// TwinCAT 3 PLC project PLC
// ProgramVersion: 3.1.4026.15
// CompilerDefines: VISU_USEPROPERTYINFO,VISU_USEWSTRING
// libraries:
//   machine_alarm_manager, * (Beckhoff Automation K.K.)
//   Tc2_MC2, * (Beckhoff Automation GmbH)
//   Tc2_Standard, * (Beckhoff Automation GmbH)
//   Tc2_System, * (Beckhoff Automation GmbH)
//   Tc2_Utilities, * (Beckhoff Automation GmbH)
//   VisuSymbols, 4.5.0.0 (System)
// project tree:
//   DUTs/ AlarmList.TcDUT, AreaStatus.TcDUT
//   / GlobalTextList.TcGTLO, PlcTask.TcTTO, Visualization Manager.TcVMO (not stored), VISU_TASK.TcTTO
//   GVLs/ GVL.TcGVL, Param.TcGVL
//   POUs/ AlarmManager.TcPOU, FB_DelaySampling.TcPOU, FB_MovingAverage.TcPOU, MAIN.TcPOU
//   VISUs/ current.TcVIS, history.TcVIS, languages.TcTLO, main.TcVIS, Visualization.TcVIS
// real-time tasks:
//   TASK PlcTask: cycle T#10ms, priority 20, ADS port 350
//   TASK VISU_TASK: cycle T#100000us, priority 30, ADS port 351
// motion (NC):
//   TASK NC-Task 1 SAF: cycle T#2ms, priority 4, ADS port 501
//   TASK NC-Task 1 SVB: cycle T#10ms, priority 8, ADS port 511
//   AXIS Axis 1 (id 1)
//     General: UnitName=°
//     Dynamic: Acceleration=1769.307, Deceleration=1769.307, Jerk=5307.921
//     Velo: RefSearch=11.79538, RefSync=11.79538, SlowManual=58.9769, FastManual=353.8614, Fast=1179.538, Maximum=1179.538
//     OtherSettings: AllowMotionCmdToSlave=true
//     encoder EncType=19
//       EncPara: ScaleFactorNumerator=360, ScaleFactorDenominator=10485760, MaxCount=#xffffffff
//     drive DrvType=16
//       DrvPara: MaxCount=#xffffffff, DriveControlDWord=#x00020100
//         Analog: VeloReferenz=1297.4918, VeloScale=32, TorqueSetpointScale=10, ScaleFactorActTorque=0.1
//         TimeComp: TaskDelayCycles=1
//     controller CtrType=1
//       CtrPara: PriorControlFactor=1
//         Observer: BandWidth=20
//   AXIS Axis 2 (id 2)
//     General: UnitName=°
//     Dynamic: Acceleration=1769.307, Deceleration=1769.307, Jerk=5307.921
//     Velo: RefSearch=11.79538, RefSync=11.79538, SlowManual=58.9769, FastManual=353.8614, Fast=1179.538, Maximum=1179.538
//     OtherSettings: AllowMotionCmdToSlave=true
//     encoder EncType=19
//       EncPara: ScaleFactorNumerator=360, ScaleFactorDenominator=10485760, MaxCount=#xffffffff
//     drive DrvType=16
//       DrvPara: MaxCount=#xffffffff, DriveControlDWord=#x00020100
//         Analog: VeloReferenz=1297.4918, VeloScale=32, TorqueSetpointScale=10, ScaleFactorActTorque=0.1
//         TimeComp: TaskDelayCycles=1
//     controller CtrType=1
//       CtrPara: PriorControlFactor=1
//         PosDiffControl: Enable=false
//         Observer: BandWidth=20
// I/O:
//   DEVICE Device 2 (EtherCAT), AmsNetId 5.69.67.250.3.1
//     Term 1 (EK1100) [EK1100 EtherCAT Coupler (2A E-Bus)]
//       Term 2 (EL1012) [EL1012 2Ch. Dig. Input 24V, 10µs]
//       Term 3 (EL1004) [EL1004 4Ch. Dig. Input 24V, 3ms]
//       Term 4 (EL1918) [EL1918, 8Ch. Safety Input 24V, TwinSAFE]
//         modules: Module 1 (FSOE), Module 2 (FSLOGIC)
//       Term 5 (EL2004) [EL2004 4Ch. Dig. Output 24V, 0.5A]
//       Term 6 (EL2084) [EL2084 4Ch. Dig. Output 24V, 0.5A, switching to negative]
//       Term 7 (EL5101-0090) [EL5101-0090 1Ch. Inc. Encoder 5V, TwinSAFE SC]
//         modules: Module 1 (EL5101-0090)
//       Term 8 (ELM7212-9018) [ELM7212-9018 2Ch. Servo Terminal (48 V, 4,5 A RMS, OCT, STO, Safe Motion, TwinSAFE Logic)]
//         modules: Module 1 (SAFETY)
//         startup 32785:21 := 0E01 // DRV Motor Settings Ch.1 / Commutation offset
//         startup 32785:27 := 10270000 // DRV Motor Settings Ch.1 / Motor speed limitation
//         startup 28688:11 := F90C // DRV Outputs Ch.1 / Torque limitation
//         startup 32784:19 := FD00 // DRV Amplifier Settings Ch.1 / Current loop proportional gain
//         startup 32784:18 := 0600 // DRV Amplifier Settings Ch.1 / Current loop integral time
//         startup 32784:21 := 2B000000 // DRV Amplifier Settings Ch.1 / Velocity loop proportional gain
//         startup 32784:20 := 96000000 // DRV Amplifier Settings Ch.1 / Velocity loop integral time
//         startup 33041:21 := 0E01 // DRV Motor Settings Ch.2 / Commutation offset
//         startup 33041:27 := 10270000 // DRV Motor Settings Ch.2 / Motor speed limitation
//         startup 28944:11 := F90C // DRV Outputs Ch.2 / Torque limitation
//         startup 33040:19 := FD00 // DRV Amplifier Settings Ch.2 / Current loop proportional gain
//         startup 33040:18 := 0600 // DRV Amplifier Settings Ch.2 / Current loop integral time
//         startup 33040:21 := 2B000000 // DRV Amplifier Settings Ch.2 / Velocity loop proportional gain
//         startup 33040:20 := 96000000 // DRV Amplifier Settings Ch.2 / Velocity loop integral time
//       Term 9 (EL9011) [EL9011 End Terminal]
//   DEVICE Device 1 (EtherCAT Automation Protocol), AmsNetId 5.69.67.250.2.1
//     Box 10 (Publisher)
//     Box 11 (Subscriber)
//     Box 12 (Publisher)
// variable links:
//   Device 2 (EtherCAT) <-> Device 1 (EtherCAT Automation Protocol)/Box 10 (Publisher)
//     Term 1 (EK1100)/Term 8 (ELM7212-9018)/Module 1 (SAFETY)/SAFETY FSoE Connection 3 Send Message/Message_11 <-> Pub-Var-Safety/Outputs/VarData
//   Device 2 (EtherCAT) <-> Device 1 (EtherCAT Automation Protocol)/Box 11 (Subscriber)
//     Term 1 (EK1100)/Term 8 (ELM7212-9018)/Module 1 (SAFETY)/SAFETY FSoE Connection 3 Receive Message/Message_11 <-> Sub-Var-Safety/Inputs/VarData
//   Device 2 (EtherCAT) <-> Device 2 (EtherCAT)/Term 1 (EK1100)/Term 8 (ELM7212-9018)
//     Term 1 (EK1100)/Term 4 (EL1918)/Module 1 (FSOE)/FSoE Inputs/FSOE <-> Module 1 (SAFETY)/SAFETY FSoE Connection 1 Receive Message/Message_3
//     Term 1 (EK1100)/Term 4 (EL1918)/Module 1 (FSOE)/FSoE Outputs/FSOE <-> Module 1 (SAFETY)/SAFETY FSoE Connection 1 Send Message/Message_3
//     Term 1 (EK1100)/Term 7 (EL5101-0090)/Module 1 (EL5101-0090)/TSC Inputs/TSC <-> Module 1 (SAFETY)/SAFETY FSoE Connection 2 Receive Message/Message_4
//     Term 1 (EK1100)/Term 7 (EL5101-0090)/Module 1 (EL5101-0090)/TSC Outputs/TSC <-> Module 1 (SAFETY)/SAFETY FSoE Connection 2 Send Message/Message_4
//   NC-Task 1 SAF/Axes/Axis 1 <-> Device 2 (EtherCAT)/Term 1 (EK1100)/Term 8 (ELM7212-9018)
//     Drive/Inputs/In/nDataIn1 <-> DRV Following error actual value Channel 1/Following error actual value
//     Drive/Inputs/In/nDcOutputTime <-> InfoData/DcOutputShift
//     Drive/Inputs/In/nState1 <-> DRV Statusword Channel 1/Statusword
//     Drive/Inputs/In/nState2 <-> DRV Statusword Channel 1/Statusword @bit 8
//     Drive/Inputs/In/nState4 @bit 1 <-> WcState/InputToggle0
//     Drive/Inputs/In/nState4 <-> WcState/WcState0
//     Drive/Outputs/Out/nCtrl1 <-> DRV Controlword Channel 1/Controlword
//     Drive/Outputs/Out/nCtrl2 <-> DRV Controlword Channel 1/Controlword @bit 8
//     Drive/Outputs/Out/nDataOut1 <-> DRV Target position Channel 1/Target position
//     Enc/Inputs/In/nDataIn1 <-> FB Position Channel 1/Position
//     Enc/Inputs/In/nDcInputTime <-> InfoData/DcInputShift
//     Enc/Inputs/In/nState4 @bit 1 <-> WcState/InputToggle0
//     Enc/Inputs/In/nState4 <-> WcState/WcState0
//   NC-Task 1 SAF/Axes/Axis 2 <-> Device 2 (EtherCAT)/Term 1 (EK1100)/Term 8 (ELM7212-9018)
//     Drive/Inputs/In/nDataIn1 <-> DRV Following error actual value Channel 2/Following error actual value
//     Drive/Inputs/In/nDcOutputTime <-> InfoData/DcOutputShift
//     Drive/Inputs/In/nState1 <-> DRV Statusword Channel 2/Statusword
//     Drive/Inputs/In/nState2 <-> DRV Statusword Channel 2/Statusword @bit 8
//     Drive/Inputs/In/nState4 @bit 1 <-> WcState/InputToggle0
//     Drive/Inputs/In/nState4 <-> WcState/WcState0
//     Drive/Outputs/Out/nCtrl1 <-> DRV Controlword Channel 2/Controlword
//     Drive/Outputs/Out/nCtrl2 <-> DRV Controlword Channel 2/Controlword @bit 8
//     Drive/Outputs/Out/nDataOut1 <-> DRV Target position Channel 2/Target position
//     Enc/Inputs/In/nDataIn1 <-> FB Position Channel 2/Position
//     Enc/Inputs/In/nDcInputTime <-> InfoData/DcInputShift
//     Enc/Inputs/In/nState4 @bit 1 <-> WcState/InputToggle0
//     Enc/Inputs/In/nState4 <-> WcState/WcState0
//   PLC/PLC Instance <-> Device 1 (EtherCAT Automation Protocol)/Box 11 (Subscriber)
//     PlcTask Inputs/MAIN.safety_master_station_emo <-> Sub-Var-Safety/Inputs/VarData/FSoE Data[0]
//   PLC/PLC Instance <-> Device 1 (EtherCAT Automation Protocol)/Box 12 (Publisher)
//     PlcTask Outputs/MAIN.eap_export_information <-> Pub-Var 11/Outputs/VarData
//   PLC/PLC Instance <-> Device 2 (EtherCAT)/Term 1 (EK1100)/Term 2 (EL1012)
//     PlcTask Inputs/MAIN.bWarningSigna02 <-> Channel 1/Input
//     PlcTask Inputs/MAIN.bWarningSigna0l <-> Channel 2/Input
//   PLC/PLC Instance <-> Device 2 (EtherCAT)/Term 1 (EK1100)/Term 3 (EL1004)
//     PlcTask Inputs/MAIN.bMcReset <-> Channel 1/Input
//   PLC/PLC Instance <-> Device 2 (EtherCAT)/Term 1 (EK1100)/Term 4 (EL1918)
//     PlcTask Inputs/MAIN.safety_emo[1] <-> Module 1 (FSOE)/FSoE Inputs/FSOE/FSIN Module 1.Input
//     PlcTask Inputs/MAIN.safety_emo[2] <-> Module 1 (FSOE)/FSoE Inputs/FSOE/FSIN Module 2.Input
//     PlcTask Inputs/MAIN.safety_input_collision_sensor <-> Module 1 (FSOE)/FSoE Inputs/FSOE/FSIN Module 4.Input
//   PLC/PLC Instance <-> Device 2 (EtherCAT)/Term 1 (EK1100)/Term 8 (ELM7212-9018)
//     PlcTask Inputs/MAIN.Enc2ActError <-> Module 1 (SAFETY)/SAFETY Standard Inputdata/Standard Out Var 10
//     PlcTask Inputs/MAIN.Enc2CmdError <-> Module 1 (SAFETY)/SAFETY Standard Inputdata/Standard Out Var 9
//     PlcTask Inputs/MAIN.SafetyMonitorSetSpeed <-> Module 1 (SAFETY)/SAFETY Standard Inputdata/Standard Out Var 14
//     PlcTask Inputs/MAIN.SafetyMonitorSpeed <-> Module 1 (SAFETY)/SAFETY Standard Inputdata/Standard Out Var 12
//     PlcTask Inputs/MAIN.SafetyRefMonitorSpeed <-> Module 1 (SAFETY)/SAFETY Standard Inputdata/Standard Out Var 13
//     PlcTask Outputs/MAIN.bSafetyErrAck <-> Module 1 (SAFETY)/SAFETY Standard Outputdata/Standard In Var 1
//     PlcTask Outputs/MAIN.bSafetyReset <-> Module 1 (SAFETY)/SAFETY Standard Outputdata/Standard In Var 7
//     PlcTask Outputs/MAIN.bSafetyRun <-> Module 1 (SAFETY)/SAFETY Standard Outputdata/Standard In Var 2
//     PlcTask Outputs/MAIN.diSpeedAct <-> Module 1 (SAFETY)/SAFETY Standard Outputdata/Standard In Var 6
//     PlcTask Outputs/MAIN.diSpeedCmd <-> Module 1 (SAFETY)/SAFETY Standard Outputdata/Standard In Var 8
//   PLC/PLC Instance <-> NC-Task 1 SAF/Axes/Axis 1
//     PlcTask Inputs/MAIN.stAxis[1].NcToPlc <-> Outputs/ToPlc
//     PlcTask Outputs/MAIN.stAxis[1].PlcToNc <-> Inputs/FromPlc
//   PLC/PLC Instance <-> NC-Task 1 SAF/Axes/Axis 2
//     PlcTask Inputs/MAIN.stAxis[2].NcToPlc <-> Outputs/ToPlc
//     PlcTask Outputs/MAIN.stAxis[2].PlcToNc <-> Inputs/FromPlc

CONFIGURATION PLC
    RESOURCE PLC ON TwinCAT3
        TASK PlcTask(INTERVAL := T#10ms, PRIORITY := 20);
        TASK VISU_TASK(INTERVAL := T#100000us, PRIORITY := 30);
        PROGRAM MAIN WITH PlcTask : MAIN;
        PROGRAM VisuElems_Visu_Prg WITH VISU_TASK : VisuElems.Visu_Prg;
    END_RESOURCE
END_CONFIGURATION

// ---- DUTs/AlarmList.TcDUT
{attribute 'qualified_only'}
{attribute 'strict'}
{attribute 'to_string'}
TYPE AlarmList :
(
	emergency_stop := 1,
	encoder_error,
	approach,
	proximity,
	collision
);
END_TYPE

// ---- DUTs/AreaStatus.TcDUT
{attribute 'qualified_only'}
{attribute 'strict'}
{attribute 'to_string'}
TYPE AreaStatus :
(
	Safe := 0,
	Hazard := 1,
	Warning_Level1 := 2,
	Warning_Level2 := 3
) := Safe;
END_TYPE

// ---- GVLs/GVL.TcGVL
{attribute 'qualified_only'}
VAR_GLOBAL
	 fb_alarm : ARRAY [1..AlarmEventParam.ALARM_MAX_COUNT] OF POINTER TO FB_Alarm;
END_VAR

// ---- GVLs/Param.TcGVL
{attribute 'qualified_only'}
VAR_GLOBAL CONSTANT
	NumberOfWarningArea		: INT := 2;
END_VAR

// ---- POUs/MAIN.TcPOU
PROGRAM MAIN
VAR
	
	
	stAxis				: ARRAY[1..2] OF AXIS_REF;
	fbMcPower			: ARRAY[1..2] OF MC_Power;
	fbMcReset			: ARRAY[1..2] OF MC_Reset;
	fbMcMoveVelocity	: ARRAY[1..2] OF MC_MoveVelocity;
	fbMcHalt			: ARRAY[1..2] OF MC_Halt;
	
	bPower		: BOOL;
	bRun		: BOOL;
	bStop		: BOOL;
	bMcReset		AT%I*	: BOOL;
	bSafetyReset	AT%Q*	: BOOL;
	bSafetyRun		AT%Q*	: BOOL := TRUE;
	bSafetyErrAck	AT%Q*	: BOOL;
	diSpeedAct		AT%Q*	: DINT;
	diSpeedCmd		AT%Q*	: DINT; 
	
	bWarningSigna0l		AT%I*	: BOOL;
	bWarningSigna02		AT%I*	: BOOL;
	Enc2ActError		AT%I*	: BOOL;
	Enc2CmdError		AT%I*	: BOOL;
	
	lrOverride		: LREAL := 50;
	_override		: LREAL;
	lrVelocity		: LREAL := 360;
	lrGearRate		: LREAL := 10;
	lrIncrement		: LREAL := 1048576;
	lrWheelIncrement	:LREAL;
	lrExtEncoderIncrement		: LREAL := 1000;
	
	diTaskIdx			: DINT;
	udiCycletime		: UDINT;
	udiTimeIntervel		: UDINT;
	udiCycleCount		: UDINT;
	fbDelaySampling		: FB_DelaySampling;
	fbDelaySamplingSet	: FB_DelaySampling;
	
	diPositionAct			: DINT;
	diPositionBufferAct		: DINT;
	diPositionCmd			: DINT;
	diPositionBufferCmd		: DINT;
	
	Mode	: INT;
	i		: UINT;
	//_Mode	: INT;
	//mode_change_delay_timer	: TON := (PT := T#1S);
	
	safety_input_collision_sensor AT%I* : BOOL;
	safety_master_station_emo AT%I* : BOOL;
	safety_emo AT%I* : ARRAY [1..2] OF BOOL;
	
	running_startup_delapy : TON := (PT := T#1S);
	
	eap_export_information	AT%Q* : ARRAY [0..7] OF BOOL;
	
	monitor_speed_average : FB_MovingAverage;
	monitor_refspeed_average : FB_MovingAverage;
	monitor_setspeed_average : FB_MovingAverage;

	SafetyMonitorSpeed AT%I* : DINT;
	SafetyRefMonitorSpeed AT%I* : DINT;
	SafetyMonitorSetSpeed AT%I* : DINT;
	
END_VAR


// Set override speed to 25 while 1sec after motor starting up. Otherwise safety error would occured by speed differential watching.
running_startup_delapy(IN := stAxis[1].Status.Moving);
IF running_startup_delapy.Q THEN
	_override := lrOverride;
ELSE
	_override := 30.0;
END_IF

FOR i:=1 TO 2 DO
	stAxis[i].ReadStatus();
	fbMcPower[i](
	Axis:= stAxis[i], 
	Enable:= bPower, 
	Enable_Positive:= bPower, 
	Enable_Negative:= bPower,
	Override := _override);

	fbMcHalt[i](
		Axis:= stAxis[i], 
		Execute:= bStop, 
		Deceleration:= 3600);
	
	fbMcReset[i](
		Axis:= stAxis[i], 
		Execute:= bMcReset);
	
	fbMcMoveVelocity[i](
		Axis:= stAxis[i],
		Execute:= bRun,
		Velocity:= lrVelocity, 
		//Direction:= MC_Direction.MC_Negative_Direction, 
		BufferMode:= MC_BufferMode.MC_Aborting);	
END_FOR
fbMcMoveVelocity[1].Direction := MC_Direction.MC_Negative_Direction;
fbMcMoveVelocity[2].Direction := MC_Direction.MC_Positive_Direction;

bSafetyReset := bMcReset;
bSafetyErrAck := bMcReset;
IF bMcReset THEN
	Mode := AreaStatus.Safe;
END_IF

IF NOT bWarningSigna0l THEN
	Mode := AreaStatus.Warning_Level1;
	IF NOT bWarningSigna02 THEN
		Mode := AreaStatus.Warning_Level2;
	END_IF
ELSIF (stAxis[1].NcToPlc.ErrorCode <> 0) OR (stAxis[2].NcToPlc.ErrorCode <> 0) THEN
	Mode := AreaStatus.Hazard;
ELSE
	Mode := AreaStatus.Safe;
END_IF

CASE Mode OF

	AreaStatus.Safe:
						lrOverride := 50;	
						
	AreaStatus.Warning_Level1:
						lrOverride := 25;
						
	AreaStatus.Warning_Level2:
						lrOverride := 10;
						
	AreaStatus.Hazard:
						lrOverride := 0;
	
END_CASE


lrWheelIncrement := lrIncrement * lrGearRate / 360;
diPositionAct := LREAL_TO_DINT(-1 * stAxis[1].NcToPlc.ActPos * lrWheelIncrement / lrExtEncoderIncrement);
diSpeedAct := diPositionAct - diPositionBufferAct; 
diPositionCmd := LREAL_TO_DINT(-1 * stAxis[1].NcToPlc.SetPos * lrWheelIncrement / lrExtEncoderIncrement);
diSpeedCmd := diPositionCmd - diPositionBufferCmd; 

diTaskIdx := GETCURTASKINDEXEX();
IF diTaskIdx > 0 THEN
    udiCycleTime := _TaskInfo[diTaskIdx].CycleTime;
	udiCycleCount := (udiTimeIntervel*10000) / udiCycleTime;
END_IF
fbDelaySampling(udiDelaySampling:= udiCycleCount, diData:= diPositionAct, diOutData=> diPositionBufferAct);
fbDelaySamplingSet(udiDelaySampling:= udiCycleCount, diData:= diPositionCmd, diOutData=> diPositionBufferCmd);

// Alarm signal

IF AlarmManager.init THEN
	GVL.fb_alarm[AlarmList.emergency_stop]^.set_activate := NOT safety_master_station_emo OR NOT safety_emo[1] OR NOT safety_emo[2];
	GVL.fb_alarm[AlarmList.approach]^.set_activate := Mode = AreaStatus.Warning_Level1;
	GVL.fb_alarm[AlarmList.proximity]^.set_activate := Mode = AreaStatus.Warning_Level2;
	GVL.fb_alarm[AlarmList.collision]^.set_activate :=  stAxis[1].Status.Moving AND NOT safety_input_collision_sensor;
	GVL.fb_alarm[AlarmList.encoder_error]^.set_activate :=  bPower AND ( NOT Enc2ActError OR NOT Enc2CmdError );

	// Send state to CP6606 controller station
	FOR i := 0 TO 7 DO
		IF i < AlarmEventParam.ALARM_MAX_COUNT THEN
			eap_export_information[i] := GVL.fb_alarm[i + 1]^.bActive;
		END_IF
	END_FOR
	eap_export_information[5] := NOT stAxis[1].Status.Disabled;
	eap_export_information[6] := stAxis[1].Status.Moving;	
END_IF

monitor_speed_average(put := SafetyMonitorSpeed);
monitor_refspeed_average(put := SafetyRefMonitorSpeed);
monitor_setspeed_average(put := SafetyMonitorSetSpeed);

AlarmManager.reset_button_input := bMcReset;
AlarmManager();

END_PROGRAM

// ---- POUs/FB_DelaySampling.TcPOU
FUNCTION_BLOCK FB_DelaySampling
VAR_INPUT
	udiDelaySampling	: UDINT;
	diData				: DINT;
END_VAR
VAR_OUTPUT
	diOutData		: DINT;
END_VAR
VAR
	i				: UDINT;
	diDelayData		: ARRAY[0..1000] OF DINT;
END_VAR

//Get latest data
diDelayData[0]:=diData;

//Slide window
FOR i:=udiDelaySampling TO 1 BY -1 DO
	diDelayData[i] := diDelayData[i -1];
END_FOR

diOutData := diDelayData[udiDelaySampling];

END_FUNCTION_BLOCK

// ---- POUs/FB_MovingAverage.TcPOU
FUNCTION_BLOCK FB_MovingAverage
VAR_INPUT
	put : DINT;
END_VAR
VAR_OUTPUT
	get : DINT;
END_VAR
VAR
	//buffer : ARRAY [1..1024] OF DINT;
	//i : UINT;
	tmp : LREAL;
	data_count : LREAL;
END_VAR

IF data_count < 16 THEN
	data_count := data_count + 1;
END_IF
tmp := (data_count * tmp + TO_LREAL(put)) / (data_count + 1);
get := TO_DINT(tmp);

END_FUNCTION_BLOCK

// ---- POUs/AlarmManager.TcPOU
PROGRAM AlarmManager
VAR_INPUT
	// input FROM HMI
	confirm_button_input		: BOOL;
	reset_button_input			: BOOL;
	history_clear_button_input	: BOOL;
END_VAR
VAR_OUTPUT
	init : BOOL;	
END_VAR
VAR
(* Alarm control *)	
	// Alarm calculation function block
	i : UINT;
	
	(*User variables*)
	// User alarm event
	error_condition					: BOOL;
	warning_condition				: BOOL;
	info_condition					: BOOL;

	error_argument				: INT := 0;
	error_code_random			: DRAND; 


	history_clear_delay_timer	: TON;

	// output to HMI
	status_unconfirm				: BOOL;
	unconfirmed_count				: UDINT;
	status_active					: BOOL;
	active_count					: UDINT;
	status_resetable				: BOOL;
	blink_timer				: TON := (PT := T#0.5S);
	
	(* For Visualization *)
    bReadEvents          : BOOL;
	
	(*Listener*)
	fb_observer : FB_EventObserver;
	subject				: FB_Subject;
	event_table_view 	: FB_Tc3EventVisualizationView;
	event_iot_exporter	: FB_EventIoTExporter;		// IoT exporter
	fbGetTimeZoneInformation	: FB_GetTimeZoneInformation := (bExecute := TRUE);
	
	tmp_string : T_MaxString;
	lang_select_options : UDINT := 1;
	
	alarm_instance : REFERENCE TO FB_ALarm;
	
	(*
	eSeverity ::
	TYPE TcEventSeverity : (
		Verbose  := 0, 
		Info     := 1, 
		Warning  := 2, 
		Error    := 3, 
		Critical := 4);
	END_TYPE
	*)
	AlarmDatabase : ARRAY [1..AlarmEventParam.ALARM_MAX_COUNT] OF ST_EventMetadata := [
		(	
			nEventId := 1,				// イベントID 1 
			eSeverity := 4, 			// TcEventSeverity
			bWithConfirmation := TRUE,	// 新規アラームと確認済みアラームの区別が必要か否か
			bWithResetOperation := TRUE	// アラーム解除のリセット操作が必要か否か
		),
		(	nEventId := 2, 
			eSeverity := 3, 
			bWithConfirmation := TRUE,
			bWithResetOperation := TRUE
		),
		(	nEventId := 3, 
			eSeverity := 1, 
			bWithConfirmation := TRUE,
			bWithResetOperation := FALSE
		),
		(	nEventId := 4, 
			eSeverity := 2, 
			bWithConfirmation := TRUE,
			bWithResetOperation := FALSE
		),
		(	nEventId := 5, 
			eSeverity := 3, 
			bWithConfirmation := TRUE,
			bWithResetOperation := TRUE
		)
	];
END_VAR

(*
	FB_Observer内の FB_Alarm インスタンス配列に対して、GVL.AlarmDatabseで定義したイベントクラスの情報で紐付ける。
*)
IF NOT init THEN
	FOR i := 1 TO AlarmEventParam.ALARM_MAX_COUNT DO
		fb_observer.event_table.init_instance(
			eventClass := TC_EVENT_CLASSES.UserDefinedEventClass,
			nEventId := AlarmDatabase[i].nEventId,
			eSeverity := AlarmDatabase[i].eSeverity,
			bWithConfirmation := AlarmDatabase[i].bWithConfirmation,
			bWithResetOperation := AlarmDatabase[i].bWithResetOperation
		);
		alarm_instance REF= fb_observer.event_table.get_alarm(i);
		GVL.fb_alarm[i] := ADR(alarm_instance);
	END_FOR
	fb_observer.event_table.viewer := subject;
	subject.subscribe(event_table_view);
	subject.subscribe(event_iot_exporter);
	init := TRUE;
END_IF

//　アラームリセットボタン受付
IF reset_button_input THEN
	fb_observer.event_table.try_clear_all_alarm();
END_IF

// アラーム確認ボタン受付
IF confirm_button_input THEN
	fb_observer.event_table.confirm_all_alarm();
END_IF


// IPCのロケール設定の読み出しと、Visualization向けイベントテーブル表示FBへのタイムゾーン情報設定
IF fbGetTimeZoneInformation.bBusy THEN
	fbGetTimeZoneInformation.bExecute := FALSE;		
END_IF
fbGetTimeZoneInformation();
event_table_view.tzinfo := fbGetTimeZoneInformation.tzInfo;
event_iot_exporter.tzinfo := fbGetTimeZoneInformation.tzInfo;

// オブザーバ（監視）オブジェクトの実行
CASE lang_select_options OF
	0: fb_observer.nLangId := 1033;
	1: fb_observer.nLangId := 1041;
END_CASE
fb_observer(event_class := TC_EVENT_CLASSES.UserDefinedEventClass);

// 表示用の変数制御　（アクティブアラーム数、未確認アラーム数、ボタン点滅制御、リセット可能状態）
active_count := fb_observer.event_table.active_event_count;
status_active := active_count > 0;
unconfirmed_count := fb_observer.event_table.unconfirmed_event_count;

status_resetable := fb_observer.event_table.set_event_count = 0 AND status_active;

IF unconfirmed_count > 0 THEN
	blink_timer(IN := NOT blink_timer.Q);
	IF blink_timer.Q THEN
		status_unconfirm := NOT status_unconfirm;
	END_IF
ELSE
	status_unconfirm := status_active;
END_IF

// 履歴の消去(5秒長押し）
history_clear_delay_timer(IN := history_clear_button_input, PT := T#5S);
IF history_clear_delay_timer.Q THEN
	fb_observer.event_table.viewer.history_clear();
END_IF

END_PROGRAM

// ---- GlobalTextList.TcGTLO
TEXTLIST GlobalTextList
  811 = '"'
  183 = '%'
  95 = '%.1f'
  724 = '%d'
  626 = '%f'
  174 = '%s'
  283 = 'AMRに必要な 安全 + 制御 + ナビゲーション + IoT が1台に集約'
  253 = 'AMRに必要な 安全(PLd) + 制御 + ナビゲーション + IoT が1台に集約'
  200 = 'AMRに必要な 安全(PLd) + 制御 + ナビゲーション + IoT がIPC`ni'
  778 = 'AMRに必要な 安全(PLd) + 制御 + ナビゲーション + IoT をOne IPCに統合'
  332 = 'Area sensor'
  956 = 'Danger zone'
  367 = 'Drive'
  160 = 'EL1918'
  536 = 'EL2904'
  210 = 'EL5021\n-0090'
  444 = 'EL6910'
  347 = 'ELM7211'
  126 = 'Encoder'
  914 = 'Encoder\nsin/cos'
  633 = 'Encoder sin/cos'
  891 = 'Encodersin/cos'
  436 = 'Errorレベル'
  257 = 'FSoE'
  904 = 'ID'
  924 = 'Infoレベル'
  62 = 'IPC'
  731 = 'K1'
  988 = 'K2'
  6 = 'Label'
  886 = 'Left'
  131 = 'Left wheel'
  234 = 'LiDAR'
  792 = 'Motion error'
  656 = 'Motor'
  526 = 'NC Error'
  749 = 'Override'
  799 = 'Power'
  856 = 'Run'
  766 = 'Safety LiDAR'
  619 = 'Speed'
  876 = 'Start'
  675 = 'TwinSAFE SC'
  682 = 'Warningレベル'
  528 = 'もしくは\n安全機能付き\nモーションドライブ'
  566 = 'もしくは安全機能付き\nモーションドライブ'
  252 = 'アラーム操作履歴'
  693 = 'テキスト'
  285 = 'ブラックチャンネル'
  443 = 'メイン'
  588 = 'モータ\nケーブル'
  169 = 'モータエンコーダ'
  757 = 'モータケーブル'
  309 = 'モータシャフト'
  486 = 'リセット'
  604 = '参照エンコーダ'
  123 = '右側ホイール'
  546 = '安全入力付き\nロジック\nターミナル'
  273 = '安全入力付き\nロジックターミナルフト'
  905 = '履歴'
  714 = '履歴消去'
  369 = '左側ホイール'
  634 = '指令速度'
  906 = '日付'
  907 = '時刻'
  945 = '未確認アラーム数'
  667 = '現在'
  481 = '現在アラーム一覧'
  655 = '発生中アラーム数'
  692 = '確認'
  819 = '言語設定'
  748 = '速度偏差'
  691 = '重要度'
END_TEXTLIST

// ---- VISUs/current.TcVIS
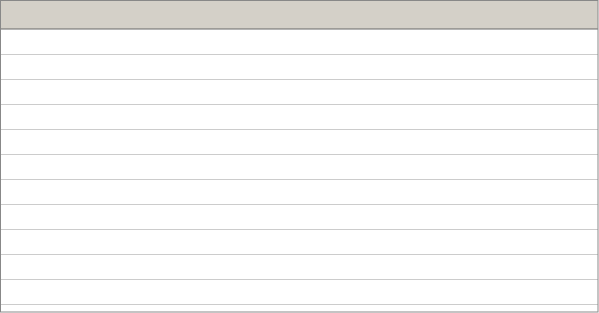
VISUALIZATION current  // 599x313
    Table (-1,-1 599x313), data array: AlarmManager.event_table_view.stAlarmEvents
        p3854506369: AlarmManager.event_table_view.stAlarmEvents[INDEX].nSourceId
        p1892666644: AlarmManager.event_table_view.stAlarmEvents[INDEX].nEventId
        p338671338: AlarmManager.event_table_view.stAlarmEvents[INDEX].Severity
        p2170511999: AlarmManager.event_table_view.stAlarmEvents[INDEX].ConfirmState
        p3723444502: AlarmManager.event_table_view.stAlarmEvents[INDEX].sDate
        p1218418051: AlarmManager.event_table_view.stAlarmEvents[INDEX].sTime
        p746581629: AlarmManager.event_table_view.stAlarmEvents[INDEX].Computer
        p3104783080: AlarmManager.event_table_view.stAlarmEvents[INDEX].sSource
        p2501879983: AlarmManager.event_table_view.stAlarmEvents[INDEX].MessageText
        p7306298: AlarmManager.event_table_view.stAlarmEvents[INDEX].bQuitMessage
        p1933151965: AlarmManager.event_table_view.stAlarmEvents[INDEX].bConfirmable
        p1755163831: 重要度
        p4092479075: 確認
        p2237128397: 日付
        p505689113: 時刻
        p2243050616: テキスト
        p1014161805: AlarmManager.event_table_view.DISP_ROWS - 1 + INT#1
END_VISUALIZATION

// ---- VISUs/history.TcVIS
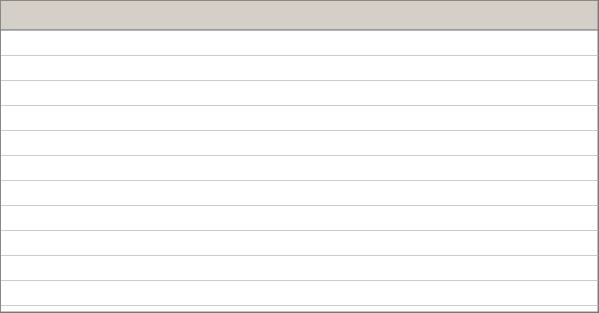
VISUALIZATION history  // 599x313
    Table (0,0 599x313), data array: AlarmManager.event_table_view.stAlarmhistory
        p3854506369: AlarmManager.event_table_view.stAlarmhistory[INDEX].nSourceId
        p1892666644: AlarmManager.event_table_view.stAlarmhistory[INDEX].nEventId
        p338671338: AlarmManager.event_table_view.stAlarmhistory[INDEX].Severity
        p2170511999: AlarmManager.event_table_view.stAlarmhistory[INDEX].ConfirmState
        p3723444502: AlarmManager.event_table_view.stAlarmhistory[INDEX].sDate
        p1218418051: AlarmManager.event_table_view.stAlarmhistory[INDEX].sTime
        p746581629: AlarmManager.event_table_view.stAlarmhistory[INDEX].Computer
        p3104783080: AlarmManager.event_table_view.stAlarmhistory[INDEX].sSource
        p2501879983: AlarmManager.event_table_view.stAlarmhistory[INDEX].MessageText
        p7306298: AlarmManager.event_table_view.stAlarmhistory[INDEX].bQuitMessage
        p1933151965: AlarmManager.event_table_view.stAlarmhistory[INDEX].bConfirmable
        p1755163831: 重要度
        p4092479075: 履歴
        p2237128397: 日付
        p505689113: 時刻
        p2243050616: テキスト
        p1014161805: AlarmManager.event_table_view.DISP_ROWS - 1 + INT#1
END_VISUALIZATION

// ---- VISUs/languages.TcTLO
TEXTLIST languages
  0 = '英語'
  1 = '日本語'
   = ''
END_TEXTLIST

// ---- VISUs/main.TcVIS
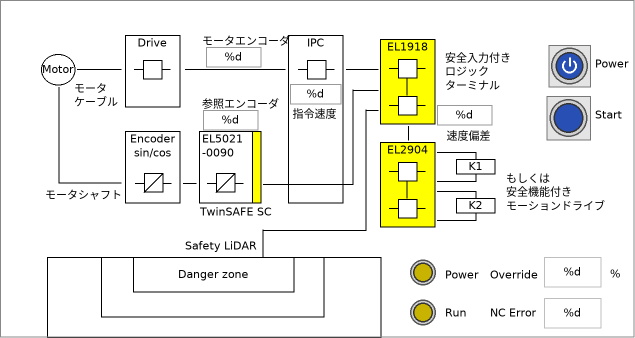
VISUALIZATION main  // 635x338
    Textfield (544,298 57x30), "%d", text variable: MAIN.stAxis[1].Status.ErrorID
    RoundedRectangle (47,257 334x81), colour toggle: NOT MAIN.bWarningSigna0l
    RoundedRectangle (101,257 223x60), colour toggle: NOT MAIN.bWarningSigna02
    RoundedRectangle (133,257 161x35), "Danger zone", colour toggle: NOT MAIN.safety_input_collision_sensor
    Label (592,49 43x30), "Power"
    Label (182,231 69x30), "Safety LiDAR"
    PowerSwitch (545,45 49x42), variable: MAIN.bPower, behaviour: TOGGLE, style: Switch-PowerSwitch-Blue
    PushSwitch (543,96 51x44), variable: MAIN.bRun, behaviour: TAP, style: Switch-PushSwitch-Blue
    Label (592,100 38x30), "Start"
    Ellipse (41,54 34x31), "Motor", colour toggle: MAIN.stAxis[1].Status.Moving
    Rectangle (125,35 55x72), "Drive"
    Line (77,69) (121,69)
    Rectangle (125,131 55x72), "Encoder sin/cos"
    Rectangle (199,131 62x72), "EL5021 -0090"
    Rectangle (252,131 9x72)
    Rectangle (288,35 55x168), "IPC"
    Line (185,69) (285,69)
    Polyline (121,183) (59,183) (59,147) (59,125) (59,87)
    Line (183,183) (196,183)
    Polyline (263,184) (353,184) (353,126) (353,90) (378,90)
    Group (135,173 36x19)
        Line (0,10) (36,10)
        Rectangle (9,0 19x19)
        Line (9,19) (28,0)
    Group (207,173 36x19)
        Line (0,10) (36,10)
        Rectangle (9,0 19x19)
        Line (9,19) (28,0)
    Group (134,60 36x19)
        Line (0,9) (36,9)
        Rectangle (9,0 19x19)
    Group (298,60 36x19)
        Line (0,9) (36,9)
        Rectangle (9,0 19x19)
    Line (346,69) (378,69)
    Rectangle (380,39 55x85), "EL1918"
    Group (389,59 36x19)
        Line (0,9) (36,9)
        Rectangle (9,0 19x19)
    Group (389,96 36x19)
        Line (0,9) (36,9)
        Rectangle (9,0 19x19)
    Line (407,95) (407,78)
    Label (42,180 83x30), "モータシャフト"
    Label (71,80 54x30), "モータ ケーブル"
    Label (197,197 91x30), "TwinSAFE SC"
    Label (442,298 35x30), "Run"
    Label (487,298 54x30), "NC Error"
    Lamp1 (408,297 30x31), variable: MAIN.stAxis[1].Status.Moving, style: Lamp-Lamp1-Yellow
    Textfield (544,257 57x30), "%d", text variable: MAIN.lrOverride
    Lamp1 (408,257 30x31), variable: MAIN.stAxis[1].Status.MotionState > 1, style: Lamp-Lamp1-Yellow
    Label (442,260 46x30), "Power"
    Label (487,260 54x30), "Override"
    Label (607,259 28x30), "%"
    Polyline (263,257) (263,230) (366,230) (366,110) (378,110)
    Rectangle (380,142 55x85), "EL2904"
    Group (389,162 36x19)
        Line (0,9) (36,9)
        Rectangle (9,0 19x19)
    Group (389,199 36x19)
        Line (0,9) (36,9)
        Rectangle (9,0 19x19)
    Line (407,198) (407,181)
    Line (437,152) (476,152)
    Line (437,181) (476,181)
    Line (476,181) (476,152)
    Rectangle (456,159 39x15), "K1"
    Line (437,191) (476,191)
    Line (437,220) (476,220)
    Line (476,220) (476,191)
    Rectangle (456,198 39x15), "K2"
    Line (408,126) (408,140)
    Label (442,48 91x47), "安全入力付き ロジック ターミナル"
    Label (503,163 112x58), "もしくは 安全機能付き モーションドライブ"
    Textfield (206,47 55x20), "%d", text variable: MAIN.SafetyMonitorSpeed
    Textfield (203,110 55x20), "%d", text variable: MAIN.SafetyRefMonitorSpeed
    Textfield (437,105 55x20), "%d", text variable: MAIN.SafetyMonitorSpeed - MAIN.SafetyRefMonitorSpeed
    Textfield (290,84 51x20), "%d", text variable: MAIN.monitor_setspeed_average.get
    Label (199,26 72x30), "モータエンコーダ"
    Label (199,89 72x30), "参照エンコーダ"
    Label (288,99 53x30), "指令速度"
    Label (442,123 53x26), "速度偏差"
END_VISUALIZATION

// ---- VISUs/Visualization.TcVIS
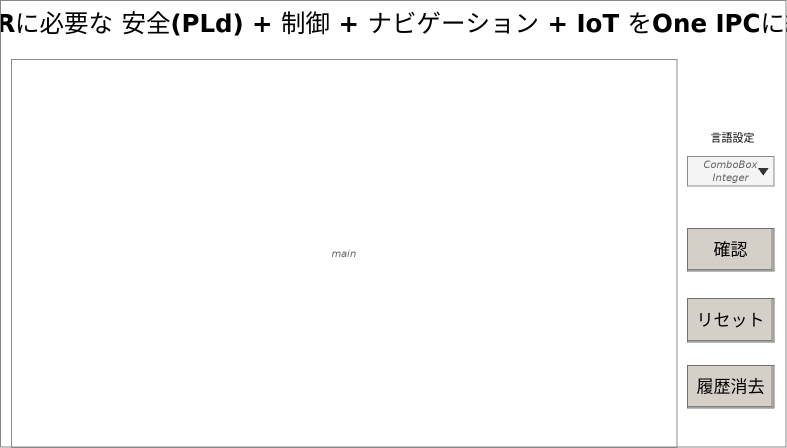
VISUALIZATION Visualization  // 787x448
    Button (687,228 87x43), "確認", colour toggle: AlarmManager.status_unconfirm
        tap AlarmManager.confirm_button_input
    Button (687,298 87x44), "リセット", colour toggle: AlarmManager.status_resetable
        tap AlarmManager.reset_button_input
    TabControl (11,59 666x389)
        shows main()
        shows current()
        shows history()
        [0]: TabTitle=メイン
        [1]: TabTitle=現在アラーム一覧
        [2]: TabTitle=アラーム操作履歴
    Label (691,121 83x34), "言語設定"
    ComboBoxInteger (687,156 87x30), variable: AlarmManager.lang_select_options, text list: 'languages'
    Button (687,365 87x43), "履歴消去"
        tap AlarmManager.history_clear_button_input
    Label (0,2 787x43), "AMRに必要な 安全(PLd) + 制御 + ナビゲーション + IoT をOne IPCに統合"
END_VISUALIZATION
